# B&R Automation Studio project AS_lab_2
Automation Studio 4.5.2.102

## Configuration Config1

### Hardware
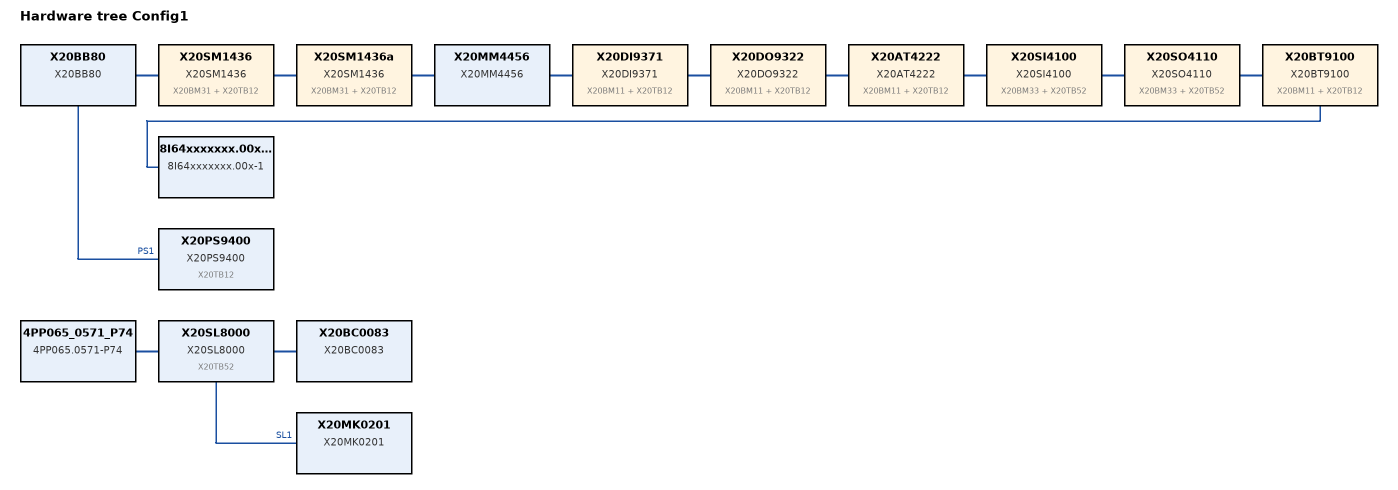
```
4PP065_0571_P74 : 4PP065.0571-P74 v1.1.2.0
  Connector IF5:
    ActivateDevice = 1
  ConfigurationID = Lab2_Config1
  TimerDeviceType = EPLX2X
  TimerDevice = 4PP065_0571_P74.IF4
  TaskClassIdleTime = 2000
  Cyclic1Duration = 2000
  Cyclic1Output = 1
8I64xxxxxxx.00x-1 : 8I64xxxxxxx.00x-1 v1.3.9.1  [X2X1 -> X20BT9100.X2X1 [Cable Type=X2XCable, Length=10, Version=1.0.0.2]]
  FunctionModel = Standard
  packedETAD = packed
  packedETI = packed
  packedCMDD = packed
  packedCMI = packed
  UNS = 220
  NCR = 10
  NSP = 890
  COS = 64
  RSC = 33000
X20AT4222 : X20AT4222 v1.2.3.0  [SS1 -> X20TB12e.SS; SL -> X20BM11b.SL1]
X20BB80 : X20BB80 v1.0.2.0
X20BC0083 : X20BC0083 v2.7.0.0  [PLK1 -> X20SL8000.PLK2 [Cable Type=PowerlinkCable, Length=10, Version=1.0.0.2]; SL -> X20BB80.SL1]
X20BM11 : X20BM11 v1.0.0.1  [X2X1 -> X20MM4456.X2X2]
X20BM11a : X20BM11 v1.0.0.1  [X2X1 -> X20BM11.X2X2]
X20BM11b : X20BM11 v1.0.0.1  [X2X1 -> X20BM11a.X2X2]
X20BM11c : X20BM11 v1.0.0.1  [X2X1 -> X20BM33a.X2X2]
X20BM31 : X20BM31 v1.0.0.1  [X2X1 -> X20BB80.IF1]
X20BM31a : X20BM31 v1.0.0.1  [X2X1 -> X20BM31.X2X2]
X20BM33 : X20BM33 v1.0.0.4  [X2X1 -> X20BM11b.X2X2]
X20BM33a : X20BM33 v1.0.0.4  [X2X1 -> X20BM33.X2X2]
X20BT9100 : X20BT9100 v1.0.3.0  [SS1 -> X20TB12f.SS; SL -> X20BM11c.SL1]
X20DI9371 : X20DI9371 v1.0.2.0  [SS1 -> X20TB12c.SS; SL -> X20BM11.SL1]
X20DO9322 : X20DO9322 v1.0.3.0  [SS1 -> X20TB12d.SS; SL -> X20BM11a.SL1]
X20MK0201 : X20MK0201 v1.0.0.0  [SL -> X20SL8000.SL1]
X20MM4456 : X20MM4456 v1.1.5.0  [X2X1 -> X20BM31a.X2X2]
X20PS9400 : X20PS9400 v1.0.2.4  [SS1 -> X20TB12.SS; PS -> X20BB80.PS1]
X20SI4100 : X20SI4100 v1.10.1.1  [SS1 -> X20TB52a.SS; SL -> X20BM33.SL1]
X20SL8000 : X20SL8000 v1.6.5.1  [PLK1 -> 4PP065_0571_P74.IF4 [Cable Type=PowerlinkCable, Length=10, Version=1.0.0.2]; PLK2 -> X20BC0083.PLK1 [Cable Type=PowerlinkCable, Length=10, Version=1.0.0.2]; SS1 -> X20TB52.SS]
  SafeProject = SafeLOGIC-1
X20SM1436 : X20SM1436 v1.4.2.1  [SS1 -> X20TB12a.SS; SL -> X20BM31.SL1]
X20SM1436a : X20SM1436 v1.4.2.1  [SS1 -> X20TB12b.SS; SL -> X20BM31a.SL1]
X20SO4110 : X20SO4110 v1.10.1.1  [SS1 -> X20TB52b.SS; SL -> X20BM33a.SL1]
  SafeModuleID = 3
X20TB12 : X20TB12 v1.0.0.0
X20TB12a : X20TB12 v1.0.0.0
X20TB12b : X20TB12 v1.0.0.0
X20TB12c : X20TB12 v1.0.0.0
X20TB12d : X20TB12 v1.0.0.0
X20TB12e : X20TB12 v1.0.0.0
X20TB12f : X20TB12 v1.0.0.0
X20TB52 : X20TB52 v1.0.0.1
X20TB52a : X20TB52 v1.0.0.1
X20TB52b : X20TB52 v1.0.0.1
```

### IoMap.iom - 4PP065_0571_P74/IoMap.iom
```iecst
VAR_CONFIG
	::Program:driveSM.state AT %IW."8I64xxxxxxx.00x-1".ETAD_Input;
	::Program:driveSM.command AT %QW."8I64xxxxxxx.00x-1".CMDD_Output;
	::Program:driveSM.speed AT %QW."8I64xxxxxxx.00x-1".LFRD_Output;
	::Program:doorSM.direction AT %IX."X20DI9371".DigitalInput01;
	::Program:doorSM.sw[3] AT %IX."X20DI9371".DigitalInput02;
	::Program:doorSM.sw[2] AT %IX."X20DI9371".DigitalInput03;
	::Program:doorSM.sw[1] AT %IX."X20DI9371".DigitalInput04;
	::Program:doorSM.sw[0] AT %IX."X20DI9371".DigitalInput05;
	::Program:ledSM.led[3] AT %QX."X20DO9322".DigitalOutput02;
	::Program:ledSM.led[2] AT %QX."X20DO9322".DigitalOutput03;
	::Program:ledSM.led[1] AT %QX."X20DO9322".DigitalOutput04;
	::Program:ledSM.led[0] AT %QX."X20DO9322".DigitalOutput05;
	::Program:driveSM.speedFeedback AT %IW."8I64xxxxxxx.00x-1".RFRD_Input;
END_VAR
```

## Logical view

### Global.var
```iecst
VAR
	count : USINT;
	ledEnable : BOOL;
END_VAR
```

### Library Logical/Libraries/DriveLib (ANSIC)

#### Types.typ - Exported data types
```iecst
TYPE
	DoorStates :
		(
		ST_INIT,
		ST_UNKNOWN,
		ST_OPEN,
		ST_CLOSE,
		ST_ACC_POS,
		ST_ACC_NEG,
		ST_POS,
		ST_NEG,
		ST_DEC_POS,
		ST_DEC_NEG
		);
END_TYPE
```

#### Constants.var - Exported constants
```iecst
VAR CONSTANT
	maxSpeed : INT := 890;
	minSpeed : INT := 89;
	maxFreq : USINT := 10;
	cycleTime : USINT := 2;
END_VAR
```

#### DriveLib.fun - Exported functions and function blocks
```iecst
FUNCTION_BLOCK DoorStateMachine
	VAR_INPUT
		state : DoorStates;
		sw1 : BOOL;
		sw2 : BOOL;
		sw3 : BOOL;
		sw4 : BOOL;
		direction : BOOL;
	END_VAR
	VAR_OUTPUT
		speed : INT;
	END_VAR
END_FUNCTION_BLOCK

FUNCTION_BLOCK DriveStateMachine
	VAR_INPUT
		state : UINT;
		enable : BOOL;
	END_VAR
	VAR_OUTPUT
		command : UINT;
		speed : INT;
	END_VAR
END_FUNCTION_BLOCK

FUNCTION_BLOCK LedStateMachine
	VAR_INPUT
		state : DoorStates;
	END_VAR
	VAR_OUTPUT
		led1 : BOOL;
		led2 : BOOL;
		led3 : BOOL;
		led4 : BOOL;
		timer : INT;
	END_VAR
END_FUNCTION_BLOCK
```

#### DoorStateMachine.c
```c
#include <bur/plctypes.h>
#ifdef __cplusplus
	extern "C"
	{
#endif
#include "DriveLib.h"
#ifdef __cplusplus
	};
#endif
/* TODO: Add your comment here */
void DoorStateMachine(struct DoorStateMachine* inst)
{
	if (state == DoorStates.ST_INIT)
	{
		inst->state = DoorStates.ST_UNKNOWN;
		inst->speed = 890;
	}
	else if (inst->state == DoorStates.ST_UNKNOWN)
	{
		if (inst->sw1 && inst->direction == 0)
		{
			inst->state = DoorStates.ST_OPEN;
			inst->speed = 0;
		}
		else if (inst->sw4 && inst->direction == 1)
		{
			inst->state = DoorStates.ST_CLOSE;
			inst->speed = 0;
		}
	}
	else if (inst->state == DoorStates.ST_OPEN)
	{
		if (inst->direction == 1)
		{
			inst->state = DoorStates.ST_ACC_POS;
			inst->speed = 890 / 9;
		}
	}
	else if (inst->state == DoorStates.ST_CLOSE)
	{
		if (inst->direction == 0)
		{
			inst->state = DoorStates.ST_ACC_NEG;
			inst->speed = -890 / 9;
		}
	}
	else if (inst->state == DoorStates.ST_ACC_POS)
	{
		if (inst->sw2)
		{
			inst->state = DoorStates.ST_POS;
			inst->speed = 890;
		}
		else if (inst->direction == 0)
		{
			inst->state = DoorStates.ST_DEC_NEG;
			inst->speed = -890 / 9;
		}
	}
	else if (inst->state == DoorStates.ST_ACC_NEG)
	{
		if (inst->sw3)
		{
			inst->state = DoorStates.ST_NEG;
			inst->speed = -890;
		}
		else if (inst->direction == 1)
		{
			inst->state = DoorStates.ST_DEC_POS;
			inst->speed = 890 / 9;
		}
	}
	else if (inst->state == DoorStates.ST_POS)
	{
		if (inst->sw3)
		{
			inst->state = DoorStates.ST_DEC_POS;
			inst->speed = 890 / 9;
		}
		else if (inst->direction == 0)
		{
			inst->state = DoorStates.ST_NEG;
			inst->speed = -890;
		}
	}
	else if (inst->state == DoorStates.ST_NEG)
	{
		if (inst->sw2)
		{
			inst->state = DoorStates.ST_DEC_NEG;
			inst->speed = -890 / 9;
		}
		else if (inst->direction == 1)
		{
			inst->state = DoorStates.ST_POS;
			inst->speed = 890;
		}
	}
	else if (inst->state == DoorStates.ST_DEC_POS)
	{
		if (inst->sw4)
		{
			inst->state = DoorStates.ST_CLOSE;
			inst->speed = 0;
		}
		else if (inst->direction == 0)
		{
			inst->state = DoorStates.ST_ACC_NEG;
			inst->speed = -890 / 9;
		}
	}
	else if (inst->state == DoorStates.ST_DEC_NEG)
	{
		if (inst->sw1)
		{
			inst->state = DoorStates.ST_OPEN;
			inst->speed = 0;
		}
		else if (inst->direction == 1)
		{
			inst->state = DoorStates.ST_ACC_POS;
			inst->speed = 890 / 9;
		}
	}
}
```

#### DriveStateMachine.c
```c
#include <bur/plctypes.h>
#ifdef __cplusplus
	extern "C"
	{
#endif
#include "DriveLib.h"
#ifdef __cplusplus
	};
#endif
/* TODO: Add your comment here */
void DriveStateMachine(struct DriveStateMachine* inst)
{
//	if (inst->state == DISABLED)
//	{
//		if (inst->enable == 1 && inst->state & 0x6F == STATE_SWITCHED_ON)
//		{
//			inst->state = STATE_SWITCHED_ON;
//			inst->command = CMD_SWITCHED_ON;
//		}
//	}
//	else if (inst->state == STATE_SWITCHED_ON)
//	{
//		if (inst->enable == 0)
//		{
//			inst->state = DISABLED;
//			inst->command = CMD_SHUTDOWN;
//		}
//		else if (inst->enable == 1 && inst->state & 0x6F == STATE_READY)
//		{
//			inst->state = STATE_READY;
//			inst->command = CMD_ENABLE;
//		}
//	}
//	else if (inst->state == STATE_READY)
//	{
//		if (inst->enable == 0)
//		{
//			inst->state = DISABLED;
//			inst->command = CMD_SHUTDOWN;
//		}
//	}
}
```

#### LedStateMachine.c
```c
#include <bur/plctypes.h>
#ifdef __cplusplus
	extern "C"
	{
#endif
#include "DriveLib.h"
#ifdef __cplusplus
	};
#endif
/* TODO: Add your comment here */
void LedStateMachine(struct LedStateMachine* inst)
{
	if (state == DoorStates.ST_INIT)
	{
		inst->led1 = inst->led2 = inst->led3 = inst->led4 = 0;
	}
	else if (inst->state == DoorStates.ST_UNKNOWN)
	{
		if (count++ % 100 == 0)
			ledEnable = !ledEnable;

		inst->led1 = inst->led2 = inst->led3 = inst->led4 = ledEnable;
	}
	else if (inst->state == DoorStates.ST_OPEN)
	{
		inst->led1 = 0;
		inst->led2 = 0;
		inst->led3 = 0;
		inst->led4 = 0;
	}
	else if (inst->state == DoorStates.ST_CLOSE)
	{
		inst->led1 = 1;
		inst->led2 = 1;
		inst->led3 = 1;
		inst->led4 = 1;
	}
	else if (inst->state == DoorStates.ST_ACC_POS)
	{
		inst->led1 = 0;
		inst->led2 = 0;
		if (count++ % (int)(1000 / (2 * 2 * 25)) == 0)  //25 Hz
			inst->led3 = !inst->led3;
		inst->led4 = 1;
	}
	else if (inst->state == DoorStates.ST_ACC_NEG)
	{
		if (inst->sw3)
		{
			inst->state = DoorStates.ST_NEG;
			inst->speed = -890;
		}
		else if (inst->direction == 1)
		{
			inst->state = DoorStates.ST_DEC_POS;
			inst->speed = 890 / 9;
		}
	}
	else if (inst->state == DoorStates.ST_POS)
	{
		if (inst->sw3)
		{
			inst->state = DoorStates.ST_DEC_POS;
			inst->speed = 890 / 9;
		}
		else if (inst->direction == 0)
		{
			inst->state = DoorStates.ST_NEG;
			inst->speed = -890;
		}
	}
	else if (inst->state == DoorStates.ST_NEG)
	{
		if (inst->sw2)
		{
			inst->state = DoorStates.ST_DEC_NEG;
			inst->speed = -890 / 9;
		}
		else if (inst->direction == 1)
		{
			inst->state = DoorStates.ST_POS;
			inst->speed = 890;
		}
	}
	else if (inst->state == DoorStates.ST_DEC_POS)
	{
		if (inst->sw4)
		{
			inst->state = DoorStates.ST_CLOSE;
			inst->speed = 0;
		}
		else if (inst->direction == 0)
		{
			inst->state = DoorStates.ST_ACC_NEG;
			inst->speed = -890 / 9;
		}
	}
	else if (inst->state == DoorStates.ST_DEC_NEG)
	{
		if (inst->sw1)
		{
			inst->state = DoorStates.ST_OPEN;
			inst->speed = 0;
		}
		else if (inst->direction == 1)
		{
			inst->state = DoorStates.ST_ACC_POS;
			inst->speed = 890 / 9;
		}
	}
}
```

#### SpeedToFreq.c - not listed in the package file held
```c
#include <bur/plctypes.h>
#ifdef __cplusplus
	extern "C"
	{
#endif
	#include "DriveLib.h"
#ifdef __cplusplus
	};
#endif
/* TODO: Add your comment here */
unsigned char SpeedToFreq(signed short speed)
{
	return maxFreq * (speed > 0 ? speed : -speed) / maxSpeed;
}
```

### Program Logical/Program

#### Variables.var
```iecst
VAR
	driveSM : DriveStateMachine;
	doorSM : DoorStateMachine;
	ledSM : LedStateMachine;
	state : DoorStates;
END_VAR
```

#### Main.c
```c
#include <bur/plctypes.h>

#ifdef _DEFAULT_INCLUDES
	#include <AsDefault.h>
#endif

void _INIT ProgramInit(void)
{

}

void _CYCLIC ProgramCyclic(void)
{
	//state handling
	if (state == DoorStates.ST_INIT)
	{
		ledSM.led1 = 0;
		ledSM.led2 = 0;
		ledSM.led3 = 0;
		ledSM.led4 = 0;
		driveS

		state = DoorStates.ST_UNKNOWN;
	}
	else if (state == DoorStates.ST_UNKNOWN)
	{
		if (count++ % 10 == 0)
			ledEnable = !ledEnable;

		ledSM.led1 = ledSM.led2 = ledSM.led3 = ledSM.led4 = ledEnable;

		if (doorSM.sw1 && doorSM.direction == 0)
			state = DoorStates.ST_OPEN;
		else if (doorSM.sw4 && doorSM.direction == 1)
			state = DoorStates.ST_CLOSE;
	}
	else if (state == DoorStates.ST_OPEN)
	{
		ledSM.led1 = 0;
		ledSM.led2 = 0;
		ledSM.led3 = 0;
		ledSM.led4 = 0;

		if (doorSM.direction == 1)
			state = DoorStates.ST_ACC_POS;
	}
	else if (state == DoorStates.ST_CLOSE)
	{
		ledSM.led1 = 1;
		ledSM.led2 = 1;
		ledSM.led3 = 1;
		ledSM.led4 = 1;

		if (doorSM.direction == 0)
			state = DoorStates.ST_ACC_NEG;
	}
	else if (state == DoorStates.ST_ACC_POS)
	{
		ledSM.led1 = 0;
		ledSM.led2 = 0;
		ledSM.led3 = 0;
		ledSM.led4 = 1;

		if (doorSM.sw2)
			state = DoorStates.ST_POS;
		else if (doorSM.direction == 0)
			state = DoorStates.ST_DEC_NEG;
	}
	else if (state == DoorStates.ST_ACC_NEG)
	{
		ledSM.led1 = 0;
		ledSM.led2 = 1;
		ledSM.led3 = 1;
		ledSM.led4 = 1;

		if (doorSM.sw3)
			state = DoorStates.ST_NEG;
		else if (doorSM.direction == 1)
			state = DoorStates.ST_DEC_POS;
	}
	else if (state == DoorStates.ST_POS)
	{
		ledSM.led1 = 0;
		ledSM.led2 = 0;
		ledSM.led3 = 1;
		ledSM.led4 = 1;

		if (doorSM.sw3)
			state = DoorStates.ST_DEC_POS;
		else if (doorSM.direction == 0)
			state = DoorStates.ST_NEG;
	}
	else if (state == DoorStates.ST_NEG)
	{
		ledSM.led1 = 0;
		ledSM.led2 = 0;
		ledSM.led3 = 1;
		ledSM.led4 = 1;

		if (doorSM.sw2)
			state = DoorStates.ST_DEC_NEG;
		else if (doorSM.direction == 1)
			state = DoorStates.ST_POS;
	}
	else if (state == DoorStates.ST_DEC_POS)
	{
		ledSM.led1 = 0;
		ledSM.led2 = 1;
		ledSM.led3 = 1;
		ledSM.led4 = 1;

		if (doorSM.sw4)
			state = DoorStates.ST_CLOSE;
		else if (doorSM.direction == 0)
			state = DoorStates.ST_ACC_NEG;
	}
	else if (state == DoorStates.ST_DEC_NEG)
	{
		ledSM.led1 = 0;
		ledSM.led2 = 0;
		ledSM.led3 = 0;
		ledSM.led4 = 1;

		if (doorSM.sw1)
			state = DoorStates.ST_OPEN;
		else if (doorSM.direction == 1)
			state = DoorStates.ST_ACC_POS;
	}
}

void _EXIT ProgramExit(void)
{

}
```
